{attribute 'GeneratedUsingTerminal: EK1122-0000-0018'}
{attribute addProperty BoxType "EK1122-0000-0018"}
{attribute addProperty Id "Beckhoff_EJ7xxxsub_EK1100EK1100_AB5A94672"}
{attribute addProperty CRC "3564710036"}
{attribute addProperty Size "2"}
TYPE Beckhoff_EJ7xxxEK1122_D4792894 EXTENDS EK1122_AB5A9467 :
STRUCT
	{attribute addProperty Name "Beckhoff_EJ7xxxsub_EK1100"}
	Beckhoff_EJ7xxxsub_EK1100 : EK1100_AB5A9467;
END_STRUCT
END_TYPE

(* stored: Version 1.2.0.0, ProductVersion 3.1.4024.9
   DUT Beckhoff_EJ7xxxEK1122_D4792894: Id {d91f36c1-a18f-484c-9ae4-2e2a2b06e7d6} *)
